(* PLC project Tc3_EventLogger.SendMessage Demo, tc3-libraries-kb TwinCAT 3.1 *)
(* stored: creationDateTime 2026-05-11T01:00:00, modificationDateTime 2026-05-11T01:00:00 *)

PROGRAM P_Demo_SendMessage
  VAR
    fbSendMessage : SendMessage;  (* Tc3_EventLogger.SendMessage 实例 *)
    arg_eventClass : GUID;  (* VAR_INPUT eventClass *)
    arg_nEventId : UDINT;  (* VAR_INPUT nEventId *)
    arg_eSeverity : TcEventSeverity;  (* VAR_INPUT eSeverity *)
    arg_ipSourceInfo : I_TcSourceInfo;  (* VAR_INPUT ipSourceInfo *)
    arg_nTimeStamp : ULINT;  (* VAR_INPUT nTimeStamp *)
    arg_ipArguments : I_TcArguments;  (* VAR_INPUT ipArguments *)
  END_VAR

            // ============================================================
// Tc3_EventLogger.SendMessage 演示程序（FB 实例）
// ============================================================
// 验证步骤：
//   1. 引用 Tc3_EventLogger（及依赖类型所在库 Tc2_System 等）
//   2. 编译 + 登录
//   3. 按 doc.md 给 arg_* 赋值
//   4. 在线监视 out_* / io_* 输出
// ============================================================

fbSendMessage(
    eventClass := arg_eventClass,
    nEventId := arg_nEventId,
    eSeverity := arg_eSeverity,
    ipSourceInfo := arg_ipSourceInfo,
    nTimeStamp := arg_nTimeStamp,
    ipArguments := arg_ipArguments
);

          
END_PROGRAM
